% RSLogix 500 project TRAFFIC.RSS, saved by version 8.30.00.16 %
PROJECT "TRAFFIC "    % processor: Bul.1763 MicroLogix 1100 Series B %

PROGRAM FILES
  LAD 2 "MAIN"  5 rungs

DATA FILES
  O0 OUTPUT  5 elements
  I1 INPUT  7 elements
  S2 STATUS  66 elements
  B3 BINARY  1 elements
  T4 TIMER  4 elements
  C5 COUNTER  1 elements
  R6 CONTROL  1 elements
  N7 INTEGER  1 elements
  F8 FLOAT  1 elements

LADDER 2 "MAIN"
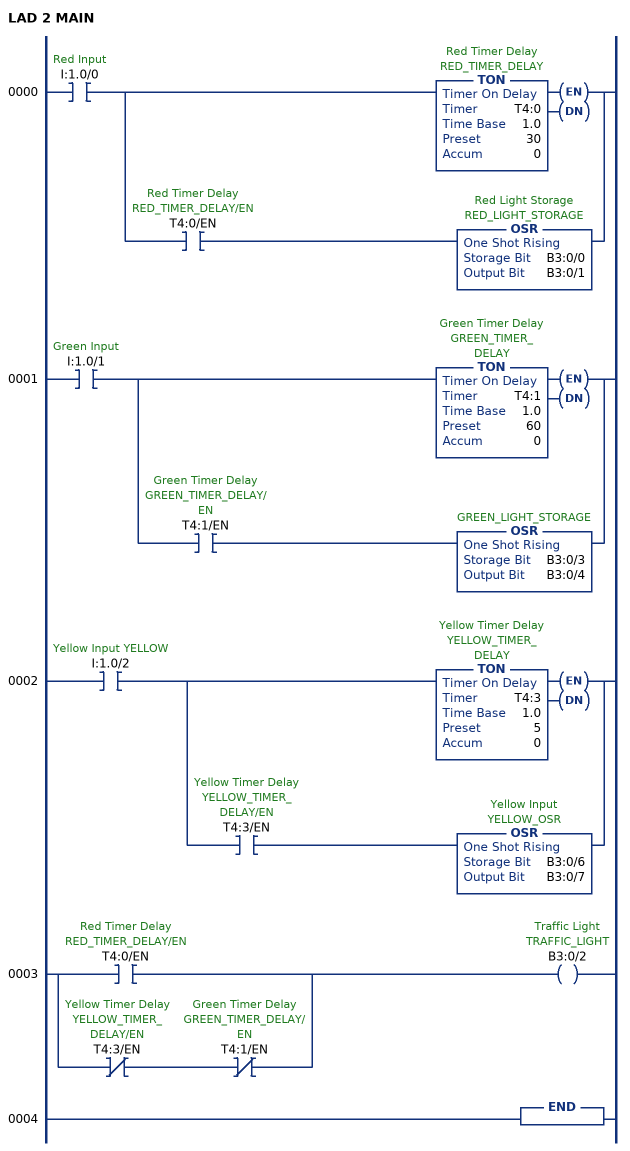
% Rung: 0 %
SOR XIC I:1.0/0 BST TON T4:0 1.0 30 0 NXB XIC T4:0/EN OSR B3:0/0 B3:0/1 BND EOR
%   I:1.0/0  "Red Input" %
%   T4:0  RED_TIMER_DELAY  "Red Timer Delay" %
%   B3:0/0  RED_LIGHT_STORAGE  "Red Light Storage" %
%   B3:0/1  "Red Light Storage OB" %
% Rung: 1 %
SOR XIC I:1.0/1 BST TON T4:1 1.0 60 0 NXB XIC T4:1/EN OSR B3:0/3 B3:0/4 BND EOR
%   I:1.0/1  "Green Input" %
%   T4:1  GREEN_TIMER_DELAY  "Green Timer Delay" %
%   B3:0/3  GREEN_LIGHT_STORAGE %
%   B3:0/4  GREEN_LIGHT_STORAGE_ %
% Rung: 2 %
SOR XIC I:1.0/2 BST TON T4:3 1.0 5 0 NXB XIC T4:3/EN OSR B3:0/6 B3:0/7 BND EOR
%   I:1.0/2  YELLOW  "Yellow Input" %
%   T4:3  YELLOW_TIMER_DELAY  "Yellow Timer Delay" %
%   B3:0/6  YELLOW_OSR  "Yellow Input" %
%   B3:0/7  "Yellow Out" %
% Rung: 3 %
SOR BST XIC T4:0/EN NXB XIO T4:3/EN XIO T4:1/EN BND OTE B3:0/2 EOR
%   T4:0  RED_TIMER_DELAY  "Red Timer Delay" %
%   T4:3  YELLOW_TIMER_DELAY  "Yellow Timer Delay" %
%   T4:1  GREEN_TIMER_DELAY  "Green Timer Delay" %
%   B3:0/2  TRAFFIC_LIGHT  "Traffic Light" %
% Rung: 4 %
SOR END EOR

OTHER DOCUMENTED ADDRESSES
  B3:0/5  GREEN_LIGHT  "Green Light"
  RED_LIGHT_SB  

DATA TABLE (non-zero values as saved)
DATA B3
% B3:0 % 0X0004
DATA T4
% .PRE .ACC %
% T4:0 % 30 0
% T4:1 % 60 0
% T4:3 % 5 0
